FUNCTION_BLOCK FB_HighLevelSystem IMPLEMENTS ITF_HighLevelSystem
VAR_INPUT
	eActivationStatus : ActivationStatus;
END_VAR
VAR_OUTPUT
END_VAR
VAR
END_VAR

PROPERTY eCondition : HighLevelCondition
GET
END_GET
END_PROPERTY

PROPERTY nErrorID : UDINT
GET
END_GET
END_PROPERTY

END_FUNCTION_BLOCK

(* stored: Version 1.1.0.1, ProductVersion 3.1.4024.12
   POU FB_HighLevelSystem: Id {f32a59e3-2d4b-4764-a617-36cef38b7412}, SpecialFunc None
   Property eCondition: Id {6df130c8-b321-441d-91d8-3607b8ea8faa}
   Get Get: Id {0fd506c0-da7e-4d3d-8a8b-1d010ebd2181}
   Property nErrorID: Id {35b6f844-4929-4eec-9295-ee6b2842d9a9}
   Get Get: Id {4338d5e2-1fec-4320-a214-083e1d5e26dc} *)
